Omron CX-Programmer project NewProject (CX-Programmer 9.75)

# PLC NewPLC1: CP1L M

## Global symbols (name address type ; comment)
0.00 BOOL  ; 灌装缸上限位
0.01 BOOL  ; 灌装缸下限位
0.02 BOOL  ; 缺瓶检测
0.03 BOOL  ; 出瓶检测
0.04 BOOL  ; 喷嘴检测
0.05 BOOL  ; 油嘴架上限位
0.06 BOOL  ; 油嘴架下限位
0.07 BOOL  ; 灌装缸原位
0.08 BOOL  ; 塞检测
0.09 BOOL  ; 中间堵瓶
0.10 BOOL  ; 星盘过载检测
0.11 BOOL  ; 星盘凸轮
100.02 BOOL  ; 进瓶阀门
100.03 BOOL  ; 出瓶阀门
100.04 BOOL  ; 夹瓶阀门
100.05 BOOL  ; 油嘴架阀门
100.06 BOOL  ; 吸盘上下阀门
100.07 BOOL  ; 吸盘前后阀门
101.00 BOOL  ; 输送带
101.01 BOOL  ; 星盘使能
101.02 BOOL  ; 真空阀门
101.03 BOOL  ; 敲塞阀门
101.04 BOOL  ; 剔除气缸
101.05 BOOL  ; 氮气阀门
1.00 BOOL  ; 门检测
1.01 BOOL  ; 加塞瓶检测
1.02 BOOL  ; 检测瓶检测
1.03 BOOL  ; 检测塞检测
1.04 BOOL  ; 剔除瓶检测
20.00 BOOL  ; 自动（触摸）
20.01 BOOL  ; 自动停（触摸）
20.04 BOOL  ; 单次灌装
20.05 BOOL  ; 灌装泵复位
20.06 BOOL  ; 装量修正
20.07 BOOL  ; 清除产量
21.00 BOOL  ; 进瓶手动
21.01 BOOL  ; 夹瓶手动
21.02 BOOL  ; 油嘴架手动
21.03 BOOL  ; 氮气手动
21.04 BOOL  ; 出瓶手动
21.05 BOOL  ; 输送带暂停
22.00 BOOL  ; 吸盘上下手动
22.01 BOOL  ; 真空手动
22.02 BOOL  ; 吸盘前后手动
22.03 BOOL  ; 敲塞手动
22.04 BOOL  ; 星盘点动
23.00 BOOL  ; 存参数
23.01 BOOL  ; 取参数
27.01 BOOL  ; 锁定
A280.04 BOOL  ; 灌装运行中
D100 CHANNEL  ; 上升加减速
D1000 CHANNEL  ; 产量
D1002 CHANNEL  ; 参数显示
D101 CHANNEL  ; 灌装上升速度
D110 CHANNEL  ; 下降加减速
D111 CHANNEL  ; 灌装缸下降速度
D120 CHANNEL  ; 复位加减速
D121 CHANNEL  ; 复位速度
D200 CHANNEL  ; 灌装脉冲数
D50 CHANNEL  ; 灌装次数
D600 CHANNEL  ; 1ml脉冲数
D6000 CHANNEL  ; 每圈装量
D6002 CHANNEL  ; 装量设定
D6003 CHANNEL  ; 实际装量
D6004 CHANNEL  ; 灌装缸上升速度
D6005 CHANNEL  ; 灌装缸下降速度
D6006 CHANNEL  ; 油嘴架延时上升
D6007 CHANNEL  ; 出瓶气缸关闭延时
D6008 CHANNEL  ; 进瓶气缸打开延时
D6009 CHANNEL  ; 灌装设定次数
D6010 CHANNEL  ; 吸盘上下延时设定
D6011 CHANNEL  ; 吸盘前/后延时设定
D6012 CHANNEL  ; 灌装头数设定
D604 CHANNEL  ; 总脉冲10倍
D608 CHANNEL  ; 总脉冲数
D612 CHANNEL  ; 实际每0.1ml脉冲数
D614 CHANNEL  ; 总脉冲10倍
D616 CHANNEL  ; 实际每圈装量
D650 CHANNEL  ; 灌装缸上升速度
D654 CHANNEL  ; 灌装缸上升速度
D660 CHANNEL  ; 灌装缸下降速度
D664 CHANNEL  ; 灌装缸下降速度
T0010 BOOL  ; 锁定时间
T0100 BOOL  ; 油嘴架下降延时
T0101 BOOL  ; 延时灌装
T0102 BOOL  ; 油嘴架延时上升
T0103 BOOL  ; 灌装结束延时
T0104 BOOL  ; 出瓶气缸延时打开
T0105 BOOL  ; 出瓶气缸关闭延时
T0106 BOOL  ; 进瓶气缸打开延时
T0107 BOOL  ; 灌装返回到位延时
T0108 BOOL  ; 进瓶气缸关闭延时
T0300 BOOL  ; 吸盘下延时
T0301 BOOL  ; 真空延时
T0302 BOOL  ; 吸盘上延时
T0303 BOOL  ; 吸盘前延时
T0304 BOOL  ; 吸盘下延时
T0305 BOOL  ; 真空释放延时
T0306 BOOL  ; 吸盘上延时
T0307 BOOL  ; 吸盘返回延时
T0500 BOOL  ; 剔除延时
W100.00 BOOL  ; 自动运行中
W100.01 BOOL  ; 停自动
W101.00 BOOL  ; 单次灌装中
W102.00 BOOL  ; 灌装泵复位中
W10.00 BOOL  ; 进瓶气缸
W10.01 BOOL  ; 夹瓶气缸
W10.02 BOOL  ; 油嘴架气缸
W10.03 BOOL  ; 氮气阀门
W10.04 BOOL  ; 出瓶气缸
W10.05 BOOL  ; 灌装泵
W200.00 BOOL  ; 星盘过载
W201.00 BOOL  ; 灌装缸上限位
W201.01 BOOL  ; 灌装缸下限位
W201.02 BOOL  ; 灌装缸原位异常
W201.03 BOOL  ; 油嘴架上限位
W201.04 BOOL  ; 油嘴架上限位
W201.05 BOOL  ; 油嘴架下限位
W201.06 BOOL  ; 灌装缸原位异常
W202.00 BOOL  ; 缺瓶报警
W202.01 BOOL  ; 中间堵瓶
W202.02 BOOL  ; 喷嘴异常
W203.00 BOOL  ; 出瓶堵
W203.01 BOOL  ; 门报警
W203.02 BOOL  ; 缺塞报警
W204.00 BOOL  ; 手动中
W204.01 BOOL  ; 自动中
W204.02 BOOL  ; 单次灌装中
W204.03 BOOL  ; 灌装泵复位中
W20.00 BOOL  ; 吸盘上下
W20.01 BOOL  ; 真空
W20.02 BOOL  ; 吸盘前后
W20.03 BOOL  ; 敲塞
W210.00 BOOL  ; 星盘过载
W210.01 BOOL  ; 灌装缸上限位
W210.02 BOOL  ; 灌装缸下限位
W210.03 BOOL  ; 灌装缸原位异常
W210.04 BOOL  ; 油嘴架上限位
W210.05 BOOL  ; 油嘴架下限位
W210.06 BOOL  ; 缺瓶报警
W210.07 BOOL  ; 中间堵瓶
W210.08 BOOL  ; 喷嘴异常
W211.00 BOOL  ; 出瓶堵
W211.01 BOOL  ; 门报警
W211.02 BOOL  ; 缺塞报警
W220.00 BOOL  ; 暂停报警条件
W220.01 BOOL  ; 灌装原位报警条件
W220.02 BOOL  ; 油嘴架上限位报警条件
W220.03 BOOL  ; 油嘴架上限位报警条件
W220.04 BOOL  ; 手动报警条件
W220.05 BOOL  ; 手动中
W220.06 BOOL  ; 自动报警条件
W220.07 BOOL  ; 单次灌装中报警条件
W220.08 BOOL  ; 灌装泵复位中报警条件
W3.00 BOOL  ; 停星盘中
W3.01 BOOL  ; 停星盘
W3.02 BOOL  ; 停自动停星盘中
W3.03 BOOL  ; 停自动停星盘
W3.04 BOOL  ; 点动停
W8.00 BOOL  ; 停输送带
出瓶堵 常开报警
单次灌装中 常开报警
灌装泵复位中 常开报警
灌装返回原位 常开报警
灌装缸上限 常闭报警
灌装缸下限 常闭报警
灌装缸原位 常闭报警
门报警 常闭报警
喷嘴异常 常闭报警
缺瓶报警 常闭报警
缺塞报警 常闭报警
手动中 常开报警
星盘过载 常开报警
油嘴架上限位 常闭报警
油嘴架上限位初始 常闭报警
油嘴架下限位 常开报警
中间堵瓶 常开报警
自动中 常开报警

## Program 新程序1 (cyclic task 0)

### Section 计算部分

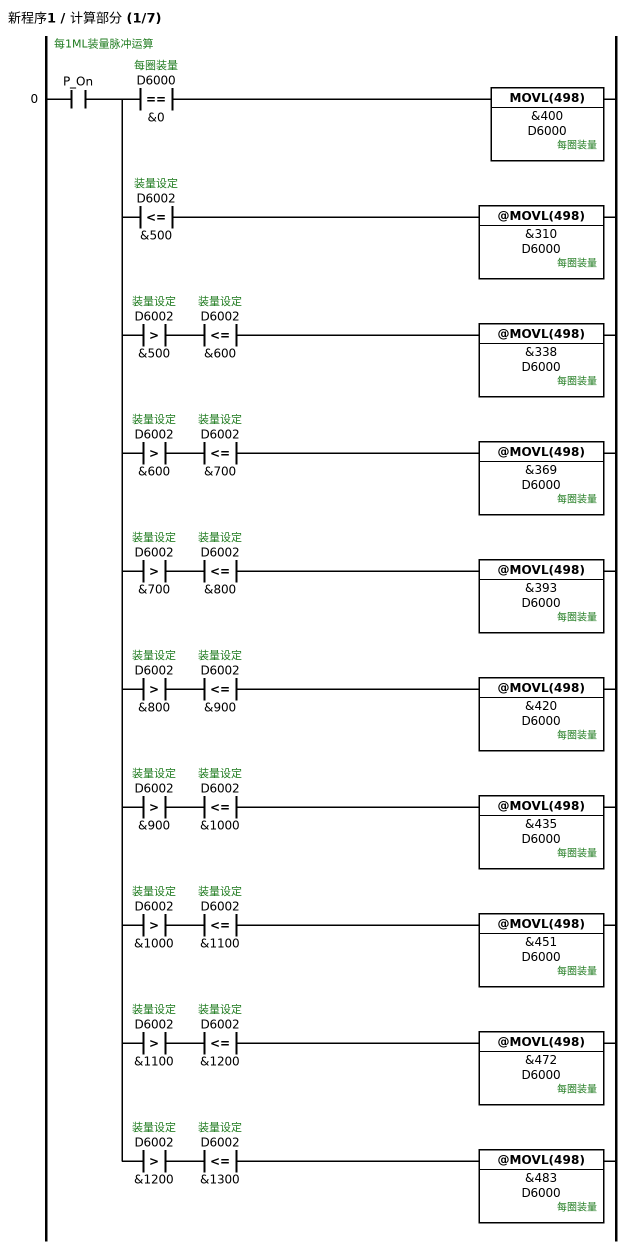
; rung 0: 每1ML装量脉冲运算
LD P_On
OUT TR0
AND=(300) D6000 &0  ; 每圈装量
MOVL(498) &400 D6000  ; 每圈装量
LD TR0
AND<=(315) D6002 &500  ; 装量设定
@MOVL(498) &310 D6000  ; 每圈装量
LD TR0
AND>(320) D6002 &500  ; 装量设定
AND<=(315) D6002 &600  ; 装量设定
@MOVL(498) &338 D6000  ; 每圈装量
LD TR0
AND>(320) D6002 &600  ; 装量设定
AND<=(315) D6002 &700  ; 装量设定
@MOVL(498) &369 D6000  ; 每圈装量
LD TR0
AND>(320) D6002 &700  ; 装量设定
AND<=(315) D6002 &800  ; 装量设定
@MOVL(498) &393 D6000  ; 每圈装量
LD TR0
AND>(320) D6002 &800  ; 装量设定
AND<=(315) D6002 &900  ; 装量设定
@MOVL(498) &420 D6000  ; 每圈装量
LD TR0
AND>(320) D6002 &900  ; 装量设定
AND<=(315) D6002 &1000  ; 装量设定
@MOVL(498) &435 D6000  ; 每圈装量
LD TR0
AND>(320) D6002 &1000  ; 装量设定
AND<=(315) D6002 &1100  ; 装量设定
@MOVL(498) &451 D6000  ; 每圈装量
LD TR0
AND>(320) D6002 &1100  ; 装量设定
AND<=(315) D6002 &1200  ; 装量设定
@MOVL(498) &472 D6000  ; 每圈装量
LD TR0
AND>(320) D6002 &1200  ; 装量设定
AND<=(315) D6002 &1300  ; 装量设定
@MOVL(498) &483 D6000  ; 每圈装量

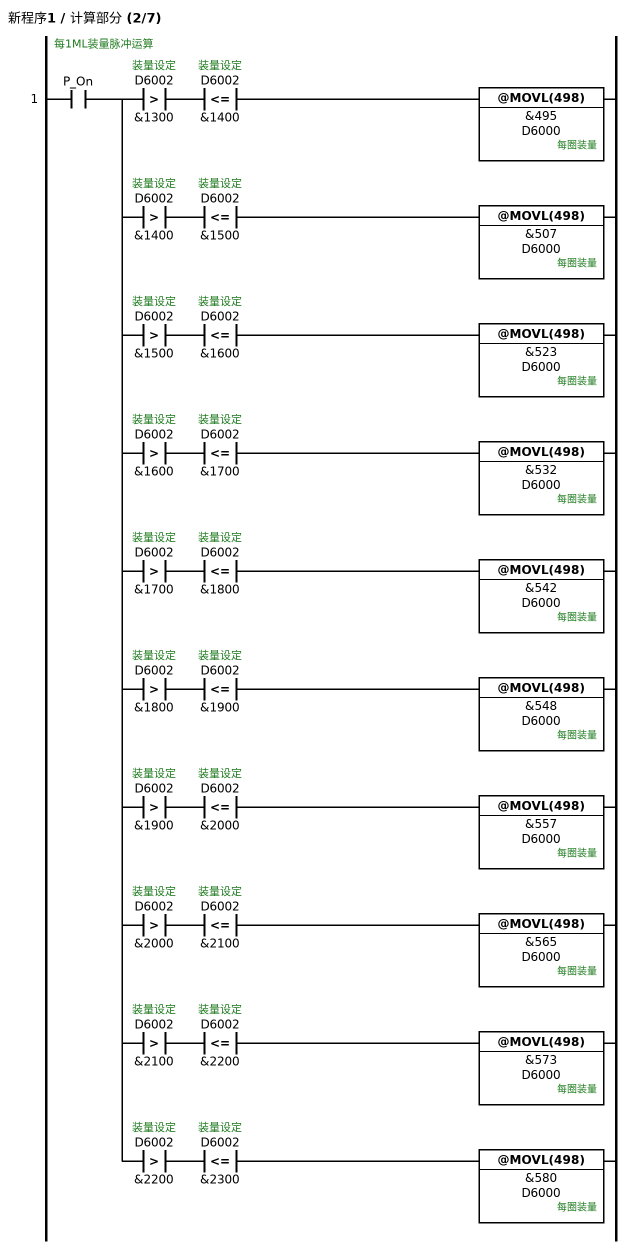
; rung 1: 每1ML装量脉冲运算
LD P_On
OUT TR0
AND>(320) D6002 &1300  ; 装量设定
AND<=(315) D6002 &1400  ; 装量设定
@MOVL(498) &495 D6000  ; 每圈装量
LD TR0
AND>(320) D6002 &1400  ; 装量设定
AND<=(315) D6002 &1500  ; 装量设定
@MOVL(498) &507 D6000  ; 每圈装量
LD TR0
AND>(320) D6002 &1500  ; 装量设定
AND<=(315) D6002 &1600  ; 装量设定
@MOVL(498) &523 D6000  ; 每圈装量
LD TR0
AND>(320) D6002 &1600  ; 装量设定
AND<=(315) D6002 &1700  ; 装量设定
@MOVL(498) &532 D6000  ; 每圈装量
LD TR0
AND>(320) D6002 &1700  ; 装量设定
AND<=(315) D6002 &1800  ; 装量设定
@MOVL(498) &542 D6000  ; 每圈装量
LD TR0
AND>(320) D6002 &1800  ; 装量设定
AND<=(315) D6002 &1900  ; 装量设定
@MOVL(498) &548 D6000  ; 每圈装量
LD TR0
AND>(320) D6002 &1900  ; 装量设定
AND<=(315) D6002 &2000  ; 装量设定
@MOVL(498) &557 D6000  ; 每圈装量
LD TR0
AND>(320) D6002 &2000  ; 装量设定
AND<=(315) D6002 &2100  ; 装量设定
@MOVL(498) &565 D6000  ; 每圈装量
LD TR0
AND>(320) D6002 &2100  ; 装量设定
AND<=(315) D6002 &2200  ; 装量设定
@MOVL(498) &573 D6000  ; 每圈装量
LD TR0
AND>(320) D6002 &2200  ; 装量设定
AND<=(315) D6002 &2300  ; 装量设定
@MOVL(498) &580 D6000  ; 每圈装量

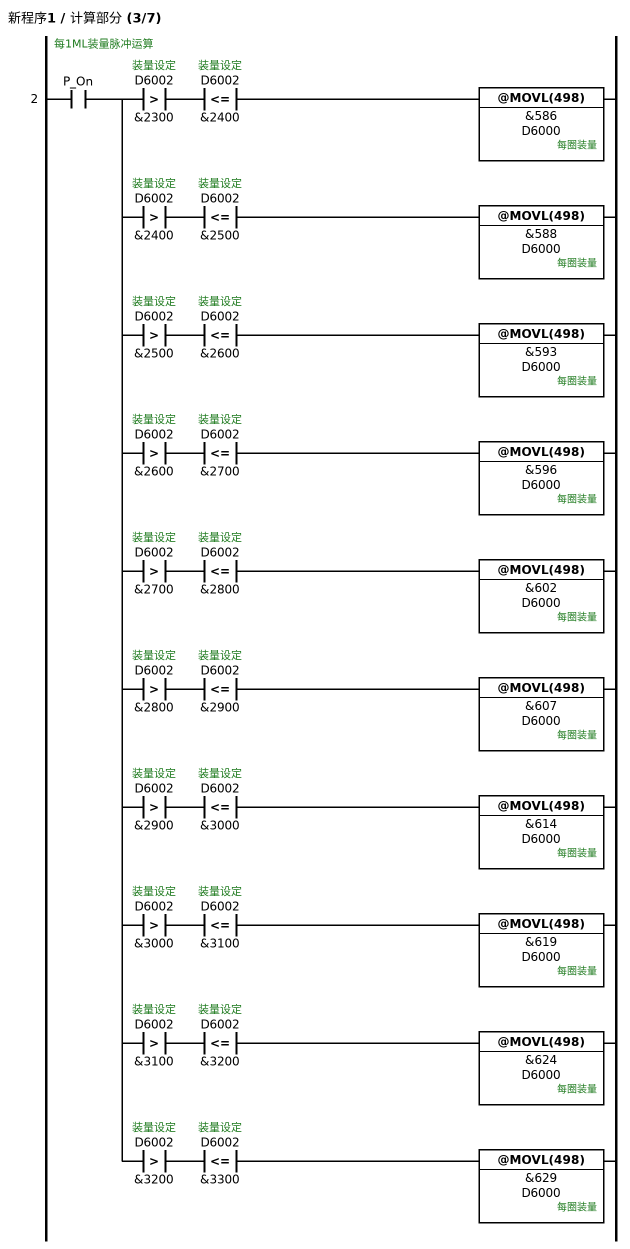
; rung 2: 每1ML装量脉冲运算
LD P_On
OUT TR0
AND>(320) D6002 &2300  ; 装量设定
AND<=(315) D6002 &2400  ; 装量设定
@MOVL(498) &586 D6000  ; 每圈装量
LD TR0
AND>(320) D6002 &2400  ; 装量设定
AND<=(315) D6002 &2500  ; 装量设定
@MOVL(498) &588 D6000  ; 每圈装量
LD TR0
AND>(320) D6002 &2500  ; 装量设定
AND<=(315) D6002 &2600  ; 装量设定
@MOVL(498) &593 D6000  ; 每圈装量
LD TR0
AND>(320) D6002 &2600  ; 装量设定
AND<=(315) D6002 &2700  ; 装量设定
@MOVL(498) &596 D6000  ; 每圈装量
LD TR0
AND>(320) D6002 &2700  ; 装量设定
AND<=(315) D6002 &2800  ; 装量设定
@MOVL(498) &602 D6000  ; 每圈装量
LD TR0
AND>(320) D6002 &2800  ; 装量设定
AND<=(315) D6002 &2900  ; 装量设定
@MOVL(498) &607 D6000  ; 每圈装量
LD TR0
AND>(320) D6002 &2900  ; 装量设定
AND<=(315) D6002 &3000  ; 装量设定
@MOVL(498) &614 D6000  ; 每圈装量
LD TR0
AND>(320) D6002 &3000  ; 装量设定
AND<=(315) D6002 &3100  ; 装量设定
@MOVL(498) &619 D6000  ; 每圈装量
LD TR0
AND>(320) D6002 &3100  ; 装量设定
AND<=(315) D6002 &3200  ; 装量设定
@MOVL(498) &624 D6000  ; 每圈装量
LD TR0
AND>(320) D6002 &3200  ; 装量设定
AND<=(315) D6002 &3300  ; 装量设定
@MOVL(498) &629 D6000  ; 每圈装量

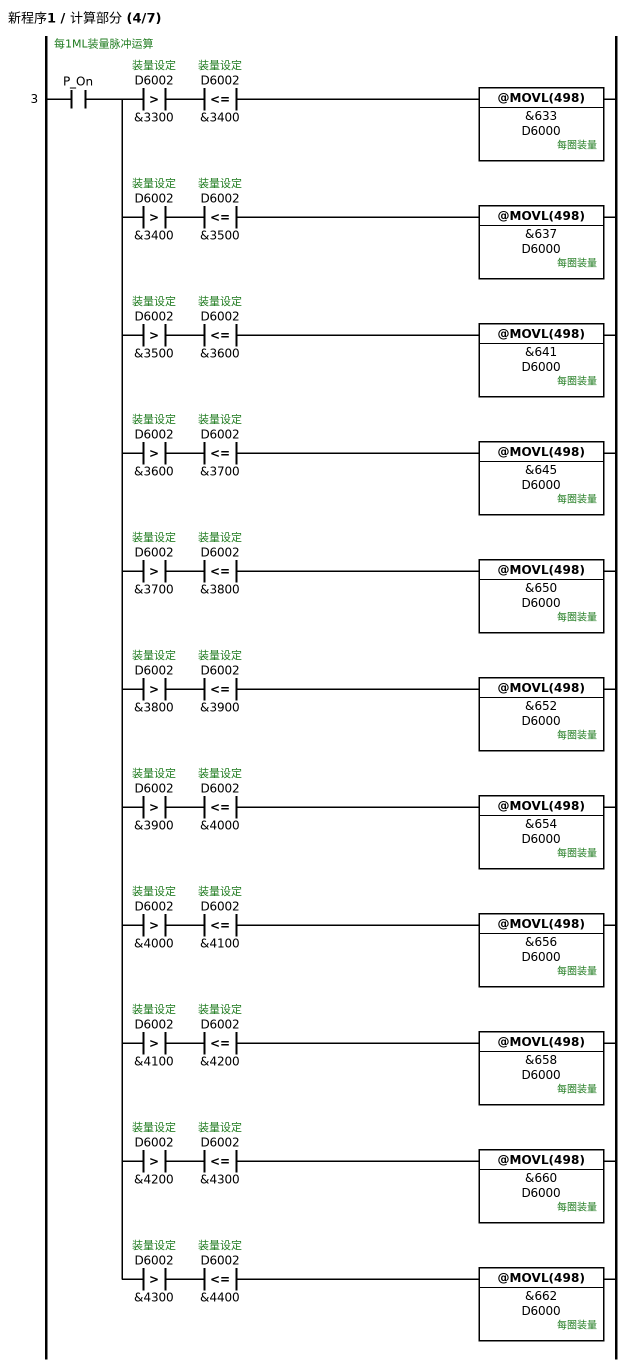
; rung 3: 每1ML装量脉冲运算
LD P_On
OUT TR0
AND>(320) D6002 &3300  ; 装量设定
AND<=(315) D6002 &3400  ; 装量设定
@MOVL(498) &633 D6000  ; 每圈装量
LD TR0
AND>(320) D6002 &3400  ; 装量设定
AND<=(315) D6002 &3500  ; 装量设定
@MOVL(498) &637 D6000  ; 每圈装量
LD TR0
AND>(320) D6002 &3500  ; 装量设定
AND<=(315) D6002 &3600  ; 装量设定
@MOVL(498) &641 D6000  ; 每圈装量
LD TR0
AND>(320) D6002 &3600  ; 装量设定
AND<=(315) D6002 &3700  ; 装量设定
@MOVL(498) &645 D6000  ; 每圈装量
LD TR0
AND>(320) D6002 &3700  ; 装量设定
AND<=(315) D6002 &3800  ; 装量设定
@MOVL(498) &650 D6000  ; 每圈装量
LD TR0
AND>(320) D6002 &3800  ; 装量设定
AND<=(315) D6002 &3900  ; 装量设定
@MOVL(498) &652 D6000  ; 每圈装量
LD TR0
AND>(320) D6002 &3900  ; 装量设定
AND<=(315) D6002 &4000  ; 装量设定
@MOVL(498) &654 D6000  ; 每圈装量
LD TR0
AND>(320) D6002 &4000  ; 装量设定
AND<=(315) D6002 &4100  ; 装量设定
@MOVL(498) &656 D6000  ; 每圈装量
LD TR0
AND>(320) D6002 &4100  ; 装量设定
AND<=(315) D6002 &4200  ; 装量设定
@MOVL(498) &658 D6000  ; 每圈装量
LD TR0
AND>(320) D6002 &4200  ; 装量设定
AND<=(315) D6002 &4300  ; 装量设定
@MOVL(498) &660 D6000  ; 每圈装量
LD TR0
AND>(320) D6002 &4300  ; 装量设定
AND<=(315) D6002 &4400  ; 装量设定
@MOVL(498) &662 D6000  ; 每圈装量

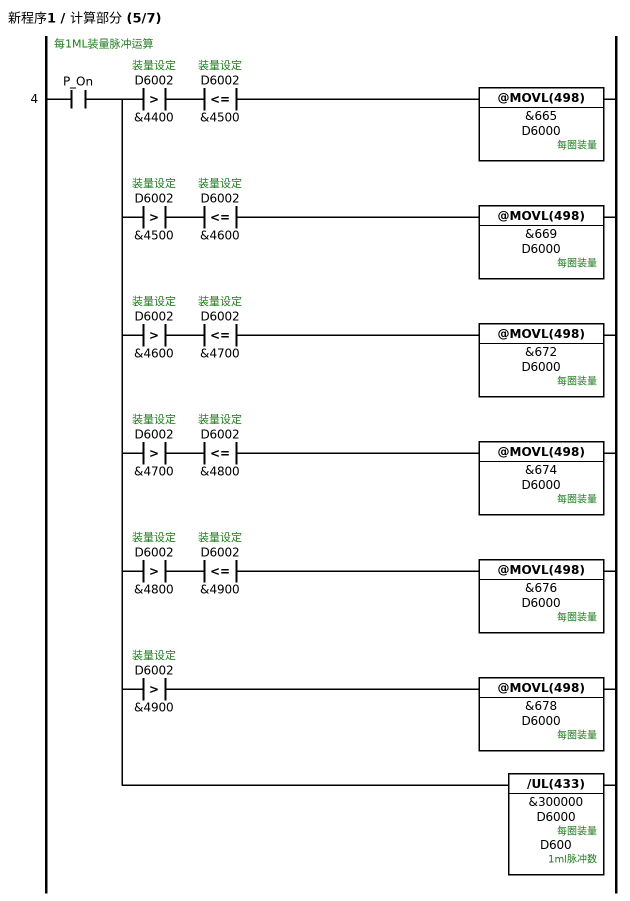
; rung 4: 每1ML装量脉冲运算
LD P_On
OUT TR0
AND>(320) D6002 &4400  ; 装量设定
AND<=(315) D6002 &4500  ; 装量设定
@MOVL(498) &665 D6000  ; 每圈装量
LD TR0
AND>(320) D6002 &4500  ; 装量设定
AND<=(315) D6002 &4600  ; 装量设定
@MOVL(498) &669 D6000  ; 每圈装量
LD TR0
AND>(320) D6002 &4600  ; 装量设定
AND<=(315) D6002 &4700  ; 装量设定
@MOVL(498) &672 D6000  ; 每圈装量
LD TR0
AND>(320) D6002 &4700  ; 装量设定
AND<=(315) D6002 &4800  ; 装量设定
@MOVL(498) &674 D6000  ; 每圈装量
LD TR0
AND>(320) D6002 &4800  ; 装量设定
AND<=(315) D6002 &4900  ; 装量设定
@MOVL(498) &676 D6000  ; 每圈装量
LD TR0
AND>(320) D6002 &4900  ; 装量设定
@MOVL(498) &678 D6000  ; 每圈装量
LD TR0
/UL(433) &300000 D6000 D600  ; 每圈装量, 1ml脉冲数

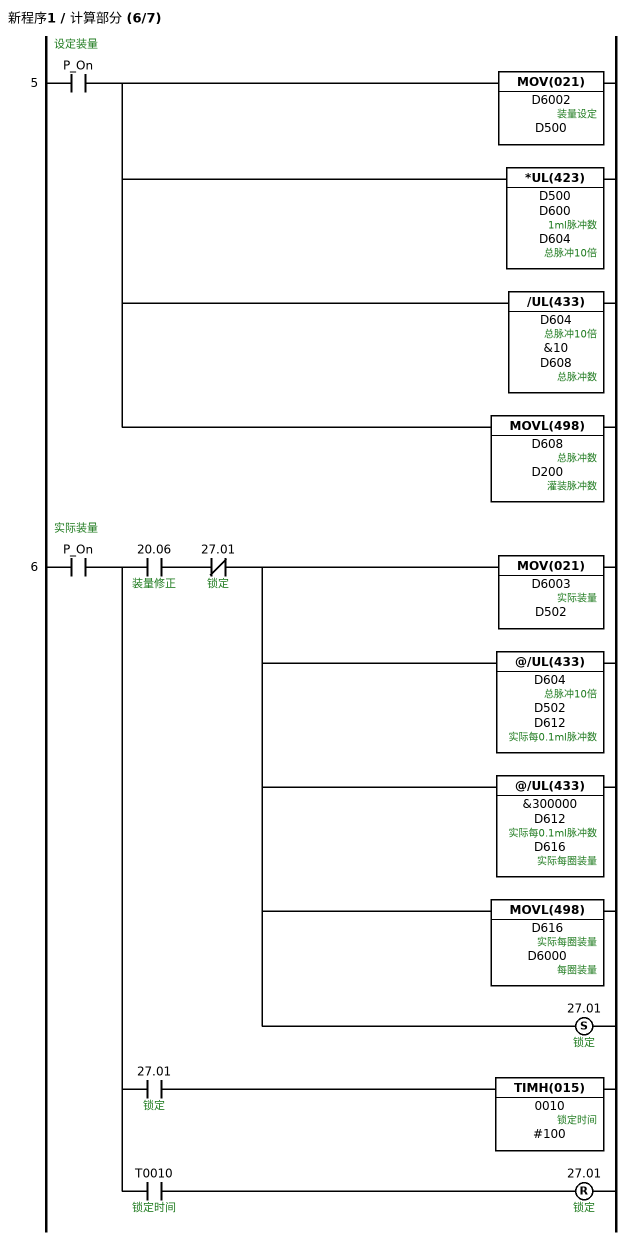
; rung 5: 设定装量
LD P_On
MOV(021) D6002 D500  ; 装量设定
*UL(423) D500 D600 D604  ; 1ml脉冲数, 总脉冲10倍
/UL(433) D604 &10 D608  ; 总脉冲10倍, 总脉冲数
MOVL(498) D608 D200  ; 总脉冲数, 灌装脉冲数
; rung 6: 实际装量
LD P_On
OUT TR0
AND 20.06  ; 装量修正
ANDNOT 27.01  ; 锁定
MOV(021) D6003 D502  ; 实际装量
@/UL(433) D604 D502 D612  ; 总脉冲10倍, 实际每0.1ml脉冲数
@/UL(433) &300000 D612 D616  ; 实际每0.1ml脉冲数, 实际每圈装量
MOVL(498) D616 D6000  ; 实际每圈装量, 每圈装量
SET 27.01  ; 锁定
LD TR0
AND 27.01  ; 锁定
TIMH(015) 0010 #100  ; 锁定时间
LD TR0
AND T0010  ; 锁定时间
RSET 27.01  ; 锁定

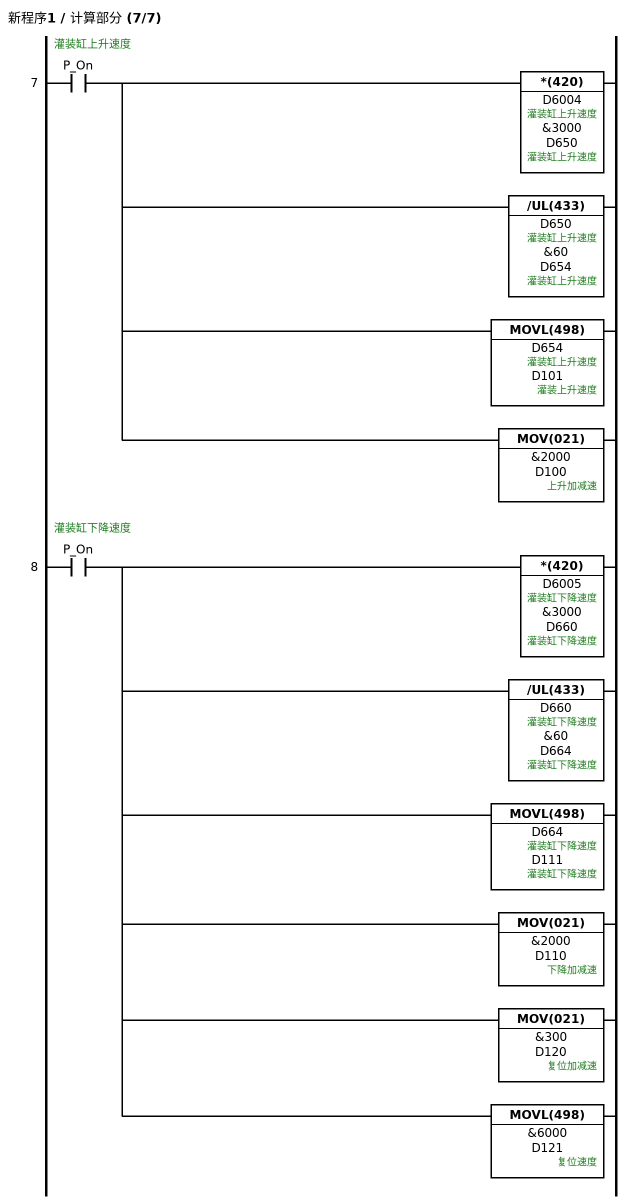
; rung 7: 灌装缸上升速度
LD P_On
*(420) D6004 &3000 D650  ; 灌装缸上升速度
/UL(433) D650 &60 D654  ; 灌装缸上升速度
MOVL(498) D654 D101  ; 灌装缸上升速度, 灌装上升速度
MOV(021) &2000 D100  ; 上升加减速
; rung 8: 灌装缸下降速度
LD P_On
*(420) D6005 &3000 D660  ; 灌装缸下降速度
/UL(433) D660 &60 D664  ; 灌装缸下降速度
MOVL(498) D664 D111  ; 灌装缸下降速度
MOV(021) &2000 D110  ; 下降加减速
MOV(021) &300 D120  ; 复位加减速
MOVL(498) &6000 D121  ; 复位速度

### Section 控制部分

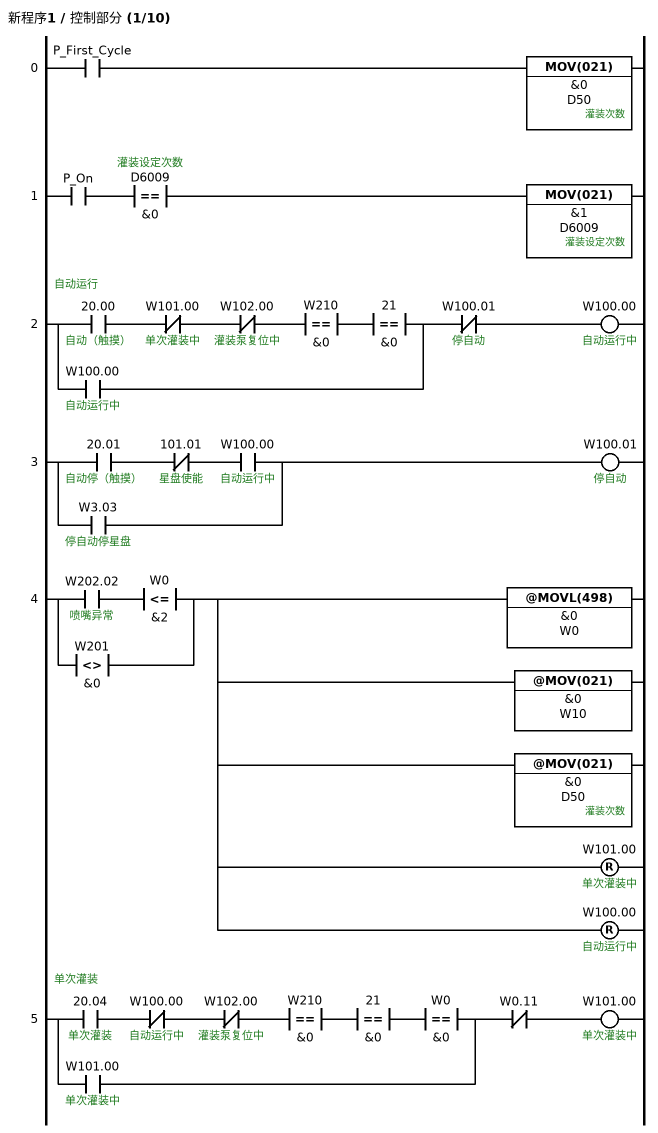
; rung 0
LD P_First_Cycle
MOV(021) &0 D50  ; 灌装次数
; rung 1
LD P_On
AND=(300) D6009 &0  ; 灌装设定次数
MOV(021) &1 D6009  ; 灌装设定次数
; rung 2: 自动运行
LD 20.00  ; 自动（触摸）
ANDNOT W101.00  ; 单次灌装中
ANDNOT W102.00  ; 灌装泵复位中
AND=L(301) W210 &0
AND=L(301) 21 &0
OR W100.00  ; 自动运行中
ANDNOT W100.01  ; 停自动
OUT W100.00  ; 自动运行中
; rung 3
LD 20.01  ; 自动停（触摸）
ANDNOT 101.01  ; 星盘使能
AND W100.00  ; 自动运行中
OR W3.03  ; 停自动停星盘
OUT W100.01  ; 停自动
; rung 4
LD W202.02  ; 喷嘴异常
AND<=(315) W0 &2
OR<>(305) W201 &0
@MOVL(498) &0 W0
@MOV(021) &0 W10
@MOV(021) &0 D50  ; 灌装次数
RSET W101.00  ; 单次灌装中
RSET W100.00  ; 自动运行中
; rung 5: 单次灌装
LD 20.04  ; 单次灌装
ANDNOT W100.00  ; 自动运行中
ANDNOT W102.00  ; 灌装泵复位中
AND=(300) W210 &0
AND=(300) 21 &0
AND=L(301) W0 &0
OR W101.00  ; 单次灌装中
ANDNOT W0.11
OUT W101.00  ; 单次灌装中

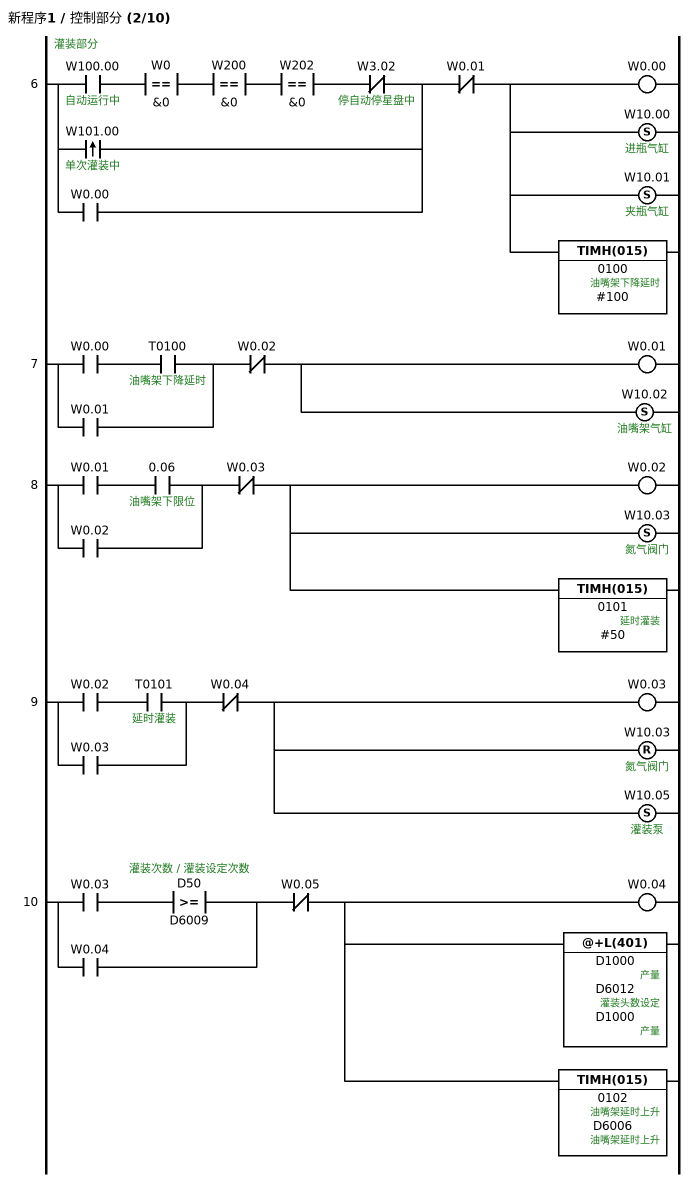
; rung 6: 灌装部分
LD W100.00  ; 自动运行中
AND=(300) W0 &0
AND=L(301) W200 &0
AND=(300) W202 &0
ANDNOT W3.02  ; 停自动停星盘中
@OR W101.00  ; 单次灌装中
OR W0.00
ANDNOT W0.01
OUT W0.00
SET W10.00  ; 进瓶气缸
SET W10.01  ; 夹瓶气缸
TIMH(015) 0100 #100  ; 油嘴架下降延时
; rung 7
LD W0.00
AND T0100  ; 油嘴架下降延时
OR W0.01
ANDNOT W0.02
OUT W0.01
SET W10.02  ; 油嘴架气缸
; rung 8
LD W0.01
AND 0.06  ; 油嘴架下限位
OR W0.02
ANDNOT W0.03
OUT W0.02
SET W10.03  ; 氮气阀门
TIMH(015) 0101 #50  ; 延时灌装
; rung 9
LD W0.02
AND T0101  ; 延时灌装
OR W0.03
ANDNOT W0.04
OUT W0.03
RSET W10.03  ; 氮气阀门
SET W10.05  ; 灌装泵
; rung 10
LD W0.03
AND>=(325) D50 D6009  ; 灌装次数, 灌装设定次数
OR W0.04
ANDNOT W0.05
OUT W0.04
@+L(401) D1000 D6012 D1000  ; 产量, 灌装头数设定
TIMH(015) 0102 D6006  ; 油嘴架延时上升

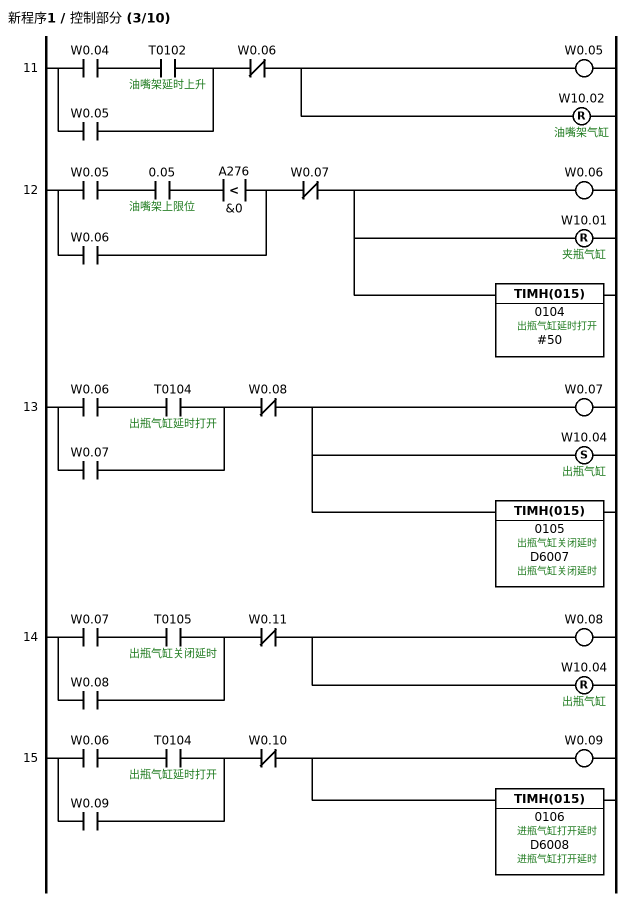
; rung 11
LD W0.04
AND T0102  ; 油嘴架延时上升
OR W0.05
ANDNOT W0.06
OUT W0.05
RSET W10.02  ; 油嘴架气缸
; rung 12
LD W0.05
AND 0.05  ; 油嘴架上限位
AND<SL(313) A276 &0
OR W0.06
ANDNOT W0.07
OUT W0.06
RSET W10.01  ; 夹瓶气缸
TIMH(015) 0104 #50  ; 出瓶气缸延时打开
; rung 13
LD W0.06
AND T0104  ; 出瓶气缸延时打开
OR W0.07
ANDNOT W0.08
OUT W0.07
SET W10.04  ; 出瓶气缸
TIMH(015) 0105 D6007  ; 出瓶气缸关闭延时
; rung 14
LD W0.07
AND T0105  ; 出瓶气缸关闭延时
OR W0.08
ANDNOT W0.11
OUT W0.08
RSET W10.04  ; 出瓶气缸
; rung 15
LD W0.06
AND T0104  ; 出瓶气缸延时打开
OR W0.09
ANDNOT W0.10
OUT W0.09
TIMH(015) 0106 D6008  ; 进瓶气缸打开延时

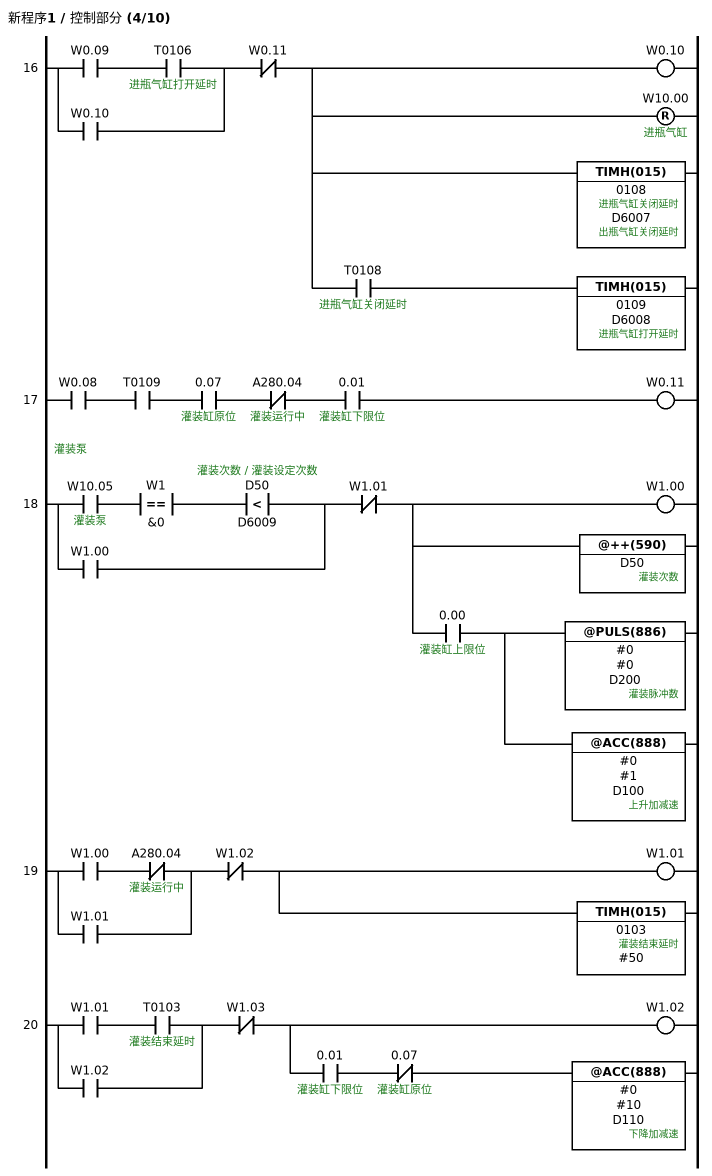
; rung 16
LD W0.09
AND T0106  ; 进瓶气缸打开延时
OR W0.10
ANDNOT W0.11
OUT W0.10
RSET W10.00  ; 进瓶气缸
TIMH(015) 0108 D6007  ; 出瓶气缸关闭延时, 进瓶气缸关闭延时
AND T0108  ; 进瓶气缸关闭延时
TIMH(015) 0109 D6008  ; 进瓶气缸打开延时
; rung 17
LD W0.08
AND T0109
AND 0.07  ; 灌装缸原位
ANDNOT A280.04  ; 灌装运行中
AND 0.01  ; 灌装缸下限位
OUT W0.11
; rung 18: 灌装泵
LD W10.05  ; 灌装泵
AND=(300) W1 &0
AND<(310) D50 D6009  ; 灌装次数, 灌装设定次数
OR W1.00
ANDNOT W1.01
OUT W1.00
@++(590) D50  ; 灌装次数
AND 0.00  ; 灌装缸上限位
@PULS(886) #0 #0 D200  ; 灌装脉冲数
@ACC(888) #0 #1 D100  ; 上升加减速
; rung 19
LD W1.00
ANDNOT A280.04  ; 灌装运行中
OR W1.01
ANDNOT W1.02
OUT W1.01
TIMH(015) 0103 #50  ; 灌装结束延时
; rung 20
LD W1.01
AND T0103  ; 灌装结束延时
OR W1.02
ANDNOT W1.03
OUT W1.02
AND 0.01  ; 灌装缸下限位
ANDNOT 0.07  ; 灌装缸原位
@ACC(888) #0 #10 D110  ; 下降加减速

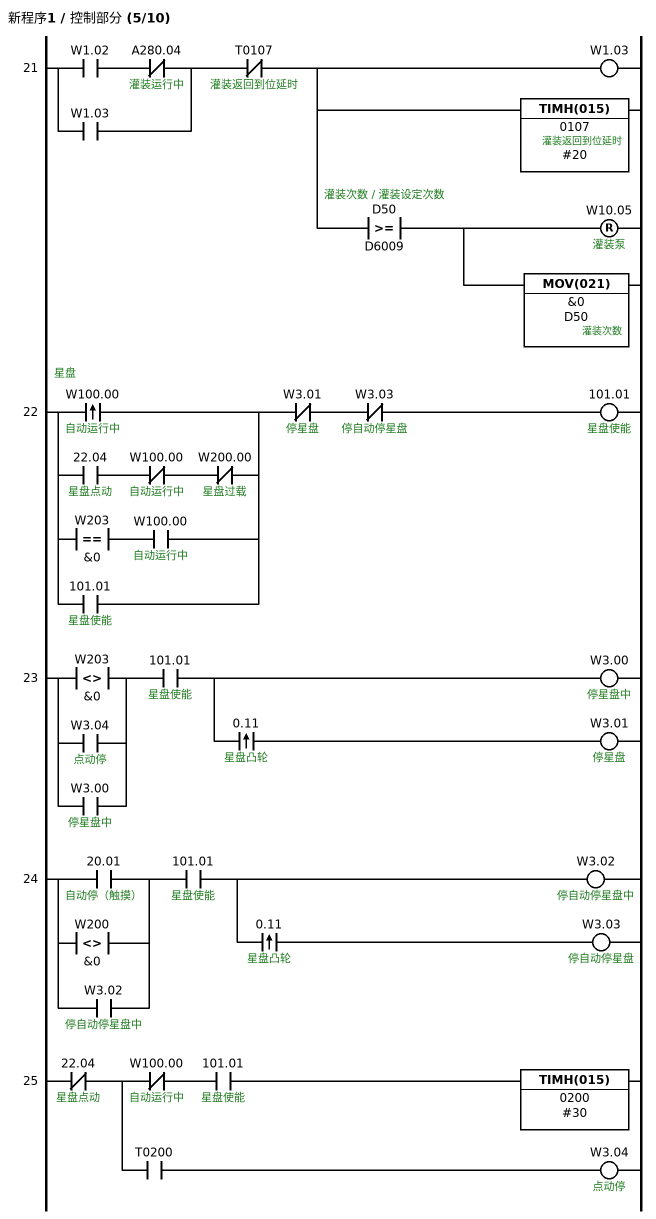
; rung 21
LD W1.02
ANDNOT A280.04  ; 灌装运行中
OR W1.03
ANDNOT T0107  ; 灌装返回到位延时
OUT W1.03
TIMH(015) 0107 #20  ; 灌装返回到位延时
AND>=(325) D50 D6009  ; 灌装次数, 灌装设定次数
RSET W10.05  ; 灌装泵
MOV(021) &0 D50  ; 灌装次数
; rung 22: 星盘
@LD W100.00  ; 自动运行中
LD 22.04  ; 星盘点动
ANDNOT W100.00  ; 自动运行中
ANDNOT W200.00  ; 星盘过载
ORLD
LD=(300) W203 &0
AND W100.00  ; 自动运行中
ORLD
OR 101.01  ; 星盘使能
ANDNOT W3.01  ; 停星盘
ANDNOT W3.03  ; 停自动停星盘
OUT 101.01  ; 星盘使能
; rung 23
LD<>(305) W203 &0
OR W3.04  ; 点动停
OR W3.00  ; 停星盘中
AND 101.01  ; 星盘使能
OUT W3.00  ; 停星盘中
@AND 0.11  ; 星盘凸轮
OUT W3.01  ; 停星盘
; rung 24
LD 20.01  ; 自动停（触摸）
OR<>L(306) W200 &0
OR W3.02  ; 停自动停星盘中
AND 101.01  ; 星盘使能
OUT W3.02  ; 停自动停星盘中
@AND 0.11  ; 星盘凸轮
OUT W3.03  ; 停自动停星盘
; rung 25
LDNOT 22.04  ; 星盘点动
OUT TR0
ANDNOT W100.00  ; 自动运行中
AND 101.01  ; 星盘使能
TIMH(015) 0200 #30
LD TR0
AND T0200
OUT W3.04  ; 点动停

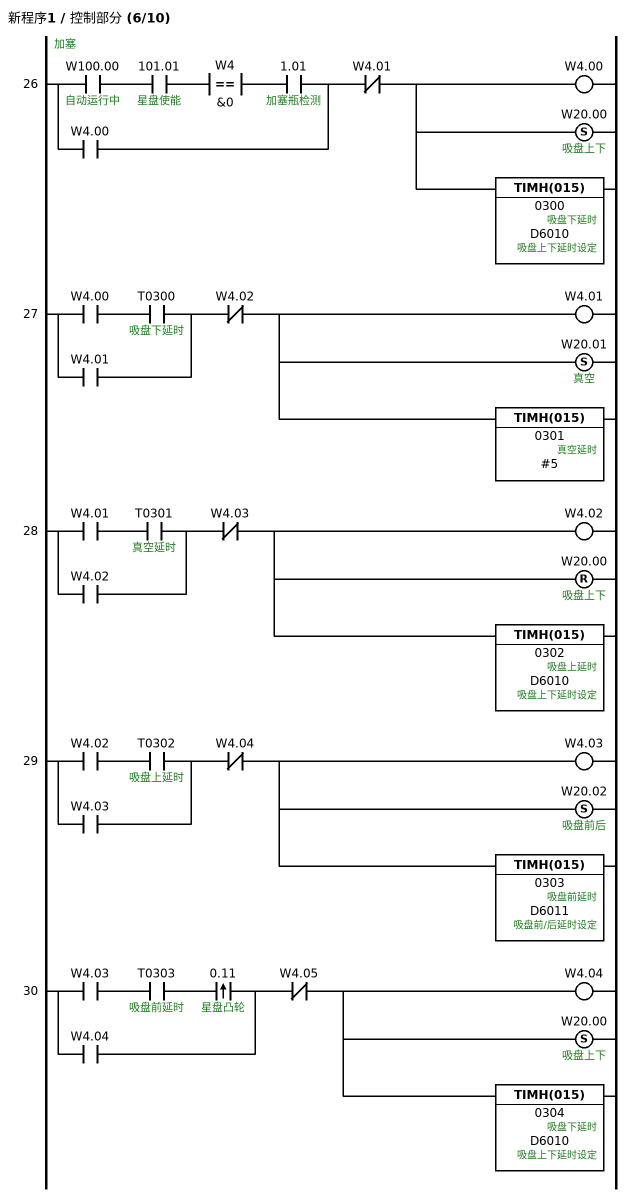
; rung 26: 加塞
LD W100.00  ; 自动运行中
AND 101.01  ; 星盘使能
AND=(300) W4 &0
AND 1.01  ; 加塞瓶检测
OR W4.00
ANDNOT W4.01
OUT W4.00
SET W20.00  ; 吸盘上下
TIMH(015) 0300 D6010  ; 吸盘上下延时设定, 吸盘下延时
; rung 27
LD W4.00
AND T0300  ; 吸盘下延时
OR W4.01
ANDNOT W4.02
OUT W4.01
SET W20.01  ; 真空
TIMH(015) 0301 #5  ; 真空延时
; rung 28
LD W4.01
AND T0301  ; 真空延时
OR W4.02
ANDNOT W4.03
OUT W4.02
RSET W20.00  ; 吸盘上下
TIMH(015) 0302 D6010  ; 吸盘上下延时设定, 吸盘上延时
; rung 29
LD W4.02
AND T0302  ; 吸盘上延时
OR W4.03
ANDNOT W4.04
OUT W4.03
SET W20.02  ; 吸盘前后
TIMH(015) 0303 D6011  ; 吸盘前/后延时设定, 吸盘前延时
; rung 30
LD W4.03
AND T0303  ; 吸盘前延时
@AND 0.11  ; 星盘凸轮
OR W4.04
ANDNOT W4.05
OUT W4.04
SET W20.00  ; 吸盘上下
TIMH(015) 0304 D6010  ; 吸盘上下延时设定, 吸盘下延时

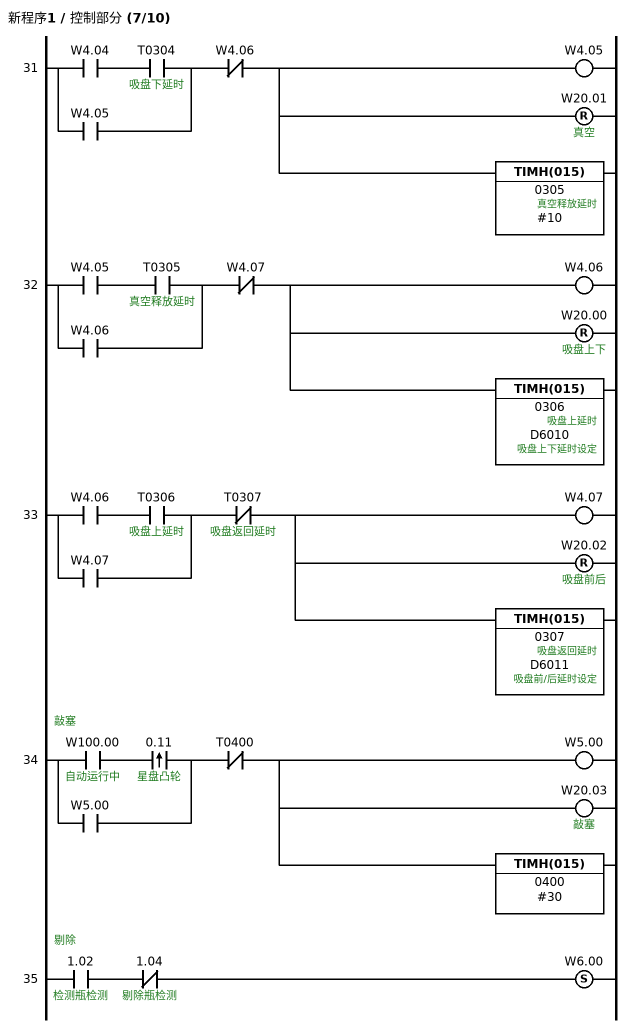
; rung 31
LD W4.04
AND T0304  ; 吸盘下延时
OR W4.05
ANDNOT W4.06
OUT W4.05
RSET W20.01  ; 真空
TIMH(015) 0305 #10  ; 真空释放延时
; rung 32
LD W4.05
AND T0305  ; 真空释放延时
OR W4.06
ANDNOT W4.07
OUT W4.06
RSET W20.00  ; 吸盘上下
TIMH(015) 0306 D6010  ; 吸盘上下延时设定, 吸盘上延时
; rung 33
LD W4.06
AND T0306  ; 吸盘上延时
OR W4.07
ANDNOT T0307  ; 吸盘返回延时
OUT W4.07
RSET W20.02  ; 吸盘前后
TIMH(015) 0307 D6011  ; 吸盘前/后延时设定, 吸盘返回延时
; rung 34: 敲塞
LD W100.00  ; 自动运行中
@AND 0.11  ; 星盘凸轮
OR W5.00
ANDNOT T0400
OUT W5.00
OUT W20.03  ; 敲塞
TIMH(015) 0400 #30
; rung 35: 剔除
LD 1.02  ; 检测瓶检测
ANDNOT 1.04  ; 剔除瓶检测
SET W6.00

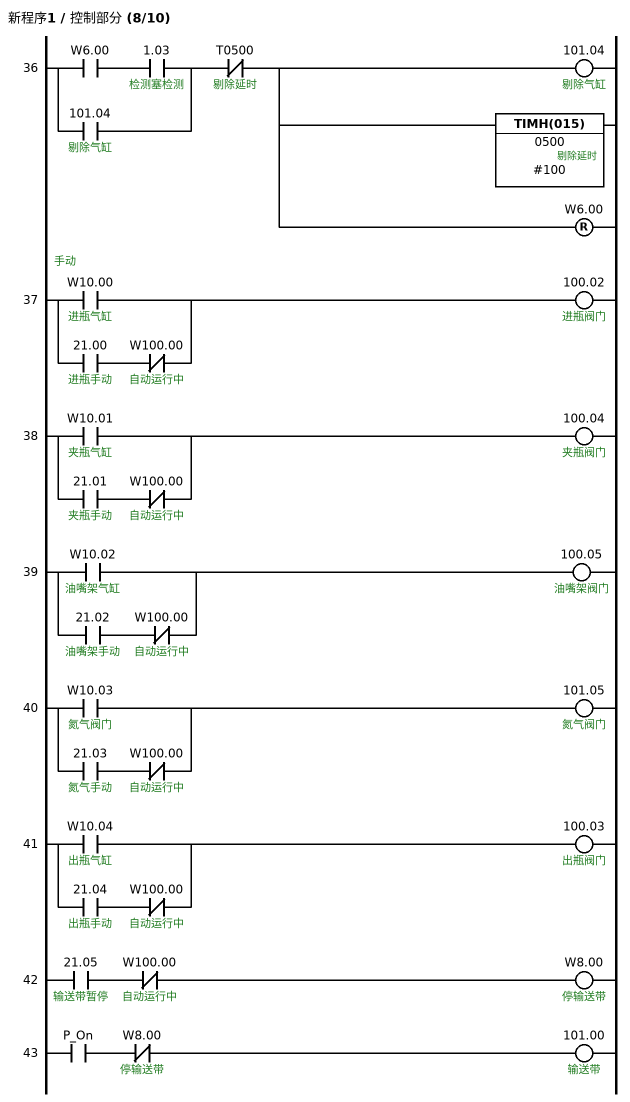
; rung 36
LD W6.00
AND 1.03  ; 检测塞检测
OR 101.04  ; 剔除气缸
ANDNOT T0500  ; 剔除延时
OUT 101.04  ; 剔除气缸
TIMH(015) 0500 #100  ; 剔除延时
RSET W6.00
; rung 37: 手动
LD W10.00  ; 进瓶气缸
LD 21.00  ; 进瓶手动
ANDNOT W100.00  ; 自动运行中
ORLD
OUT 100.02  ; 进瓶阀门
; rung 38
LD W10.01  ; 夹瓶气缸
LD 21.01  ; 夹瓶手动
ANDNOT W100.00  ; 自动运行中
ORLD
OUT 100.04  ; 夹瓶阀门
; rung 39
LD W10.02  ; 油嘴架气缸
LD 21.02  ; 油嘴架手动
ANDNOT W100.00  ; 自动运行中
ORLD
OUT 100.05  ; 油嘴架阀门
; rung 40
LD W10.03  ; 氮气阀门
LD 21.03  ; 氮气手动
ANDNOT W100.00  ; 自动运行中
ORLD
OUT 101.05  ; 氮气阀门
; rung 41
LD W10.04  ; 出瓶气缸
LD 21.04  ; 出瓶手动
ANDNOT W100.00  ; 自动运行中
ORLD
OUT 100.03  ; 出瓶阀门
; rung 42
LD 21.05  ; 输送带暂停
ANDNOT W100.00  ; 自动运行中
OUT W8.00  ; 停输送带
; rung 43
LD P_On
ANDNOT W8.00  ; 停输送带
OUT 101.00  ; 输送带

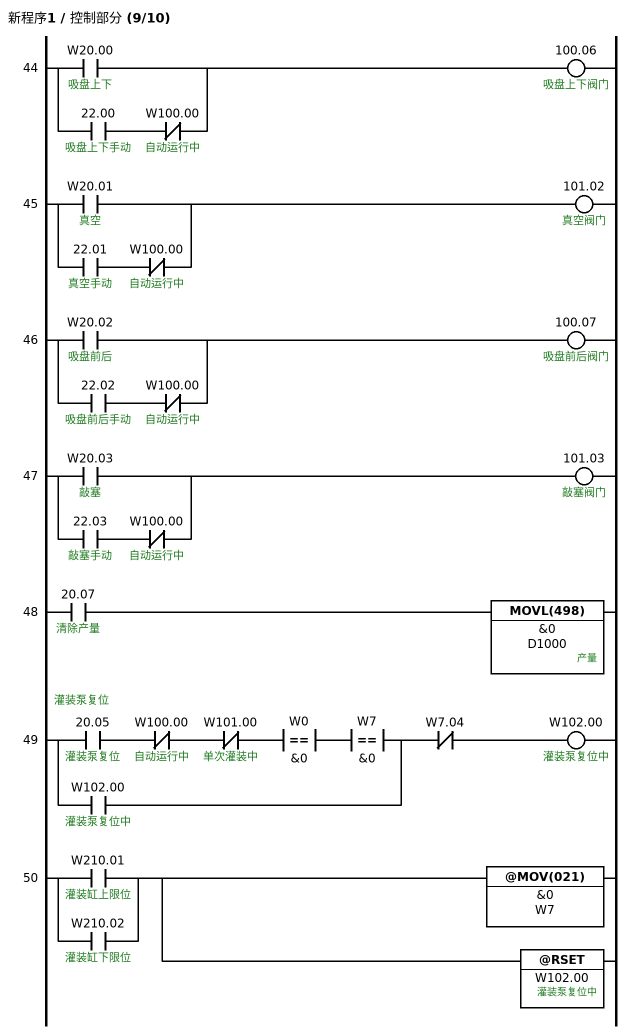
; rung 44
LD W20.00  ; 吸盘上下
LD 22.00  ; 吸盘上下手动
ANDNOT W100.00  ; 自动运行中
ORLD
OUT 100.06  ; 吸盘上下阀门
; rung 45
LD W20.01  ; 真空
LD 22.01  ; 真空手动
ANDNOT W100.00  ; 自动运行中
ORLD
OUT 101.02  ; 真空阀门
; rung 46
LD W20.02  ; 吸盘前后
LD 22.02  ; 吸盘前后手动
ANDNOT W100.00  ; 自动运行中
ORLD
OUT 100.07  ; 吸盘前后阀门
; rung 47
LD W20.03  ; 敲塞
LD 22.03  ; 敲塞手动
ANDNOT W100.00  ; 自动运行中
ORLD
OUT 101.03  ; 敲塞阀门
; rung 48
LD 20.07  ; 清除产量
MOVL(498) &0 D1000  ; 产量
; rung 49: 灌装泵复位
LD 20.05  ; 灌装泵复位
ANDNOT W100.00  ; 自动运行中
ANDNOT W101.00  ; 单次灌装中
AND=L(301) W0 &0
AND=(300) W7 &0
OR W102.00  ; 灌装泵复位中
ANDNOT W7.04
OUT W102.00  ; 灌装泵复位中
; rung 50
LD W210.01  ; 灌装缸上限位
OR W210.02  ; 灌装缸下限位
@MOV(021) &0 W7
@RSET W102.00  ; 灌装泵复位中

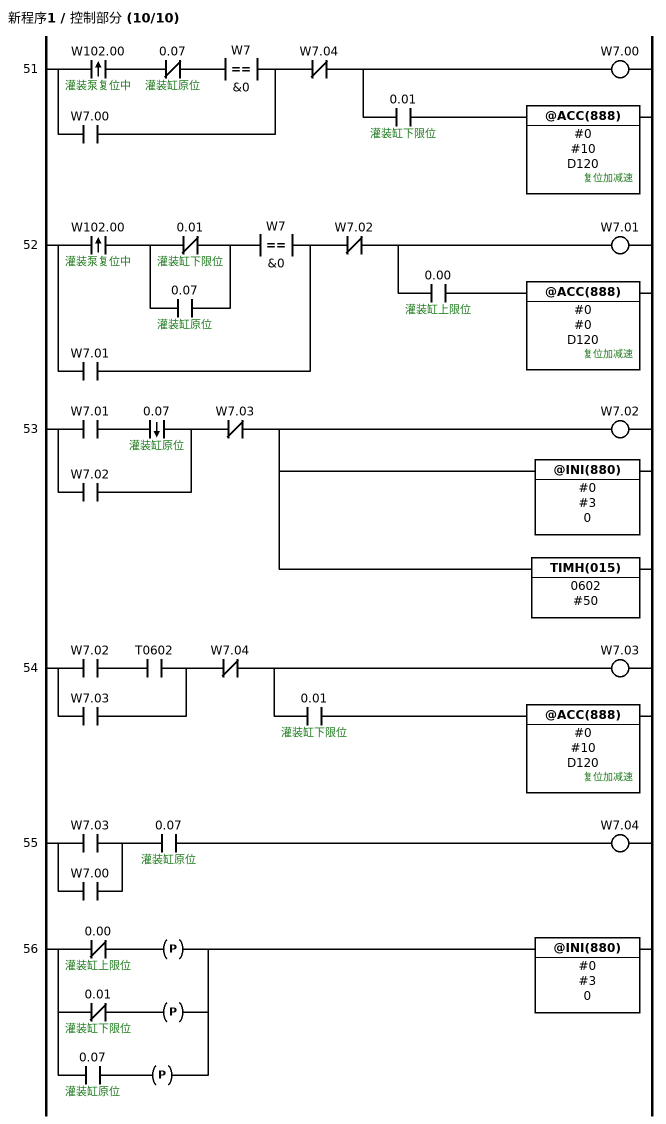
; rung 51
@LD W102.00  ; 灌装泵复位中
ANDNOT 0.07  ; 灌装缸原位
AND=(300) W7 &0
OR W7.00
ANDNOT W7.04
OUT W7.00
AND 0.01  ; 灌装缸下限位
@ACC(888) #0 #10 D120  ; 复位加减速
; rung 52
@LD W102.00  ; 灌装泵复位中
LDNOT 0.01  ; 灌装缸下限位
OR 0.07  ; 灌装缸原位
ANDLD
AND=(300) W7 &0
OR W7.01
ANDNOT W7.02
OUT W7.01
AND 0.00  ; 灌装缸上限位
@ACC(888) #0 #0 D120  ; 复位加减速
; rung 53
LD W7.01
%AND 0.07  ; 灌装缸原位
OR W7.02
ANDNOT W7.03
OUT W7.02
@INI(880) #0 #3 0
TIMH(015) 0602 #50
; rung 54
LD W7.02
AND T0602
OR W7.03
ANDNOT W7.04
OUT W7.03
AND 0.01  ; 灌装缸下限位
@ACC(888) #0 #10 D120  ; 复位加减速
; rung 55
LD W7.03
OR W7.00
AND 0.07  ; 灌装缸原位
OUT W7.04
; rung 56
LDNOT 0.00  ; 灌装缸上限位
UP(521)
LDNOT 0.01  ; 灌装缸下限位
UP(521)
ORLD
LD 0.07  ; 灌装缸原位
UP(521)
ORLD
@INI(880) #0 #3 0

### Section 报警部分

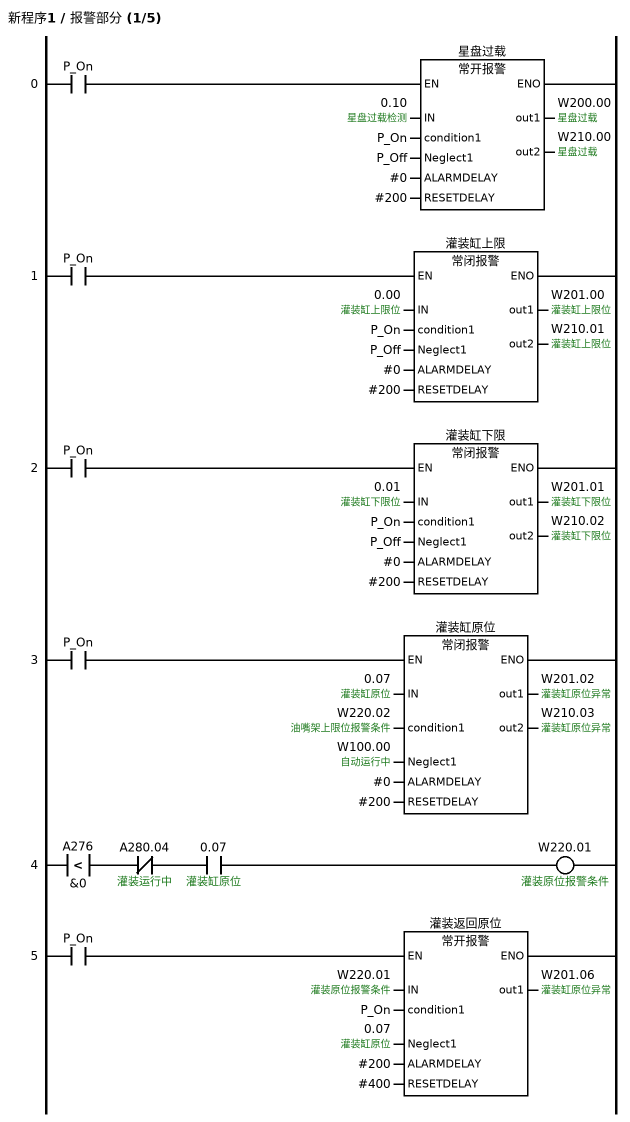
; rung 0
LD P_On
CALL 星盘过载 : 常开报警 (IN := 0.10, condition1 := P_On, Neglect1 := P_Off, ALARMDELAY := #0, RESETDELAY := #200, out1 => W200.00, out2 => W210.00)  ; 星盘过载检测, 星盘过载
; rung 1
LD P_On
CALL 灌装缸上限 : 常闭报警 (IN := 0.00, condition1 := P_On, Neglect1 := P_Off, ALARMDELAY := #0, RESETDELAY := #200, out1 => W201.00, out2 => W210.01)  ; 灌装缸上限位
; rung 2
LD P_On
CALL 灌装缸下限 : 常闭报警 (IN := 0.01, condition1 := P_On, Neglect1 := P_Off, ALARMDELAY := #0, RESETDELAY := #200, out1 => W201.01, out2 => W210.02)  ; 灌装缸下限位
; rung 3
LD P_On
CALL 灌装缸原位 : 常闭报警 (IN := 0.07, condition1 := W220.02, Neglect1 := W100.00, ALARMDELAY := #0, RESETDELAY := #200, out1 => W201.02, out2 => W210.03)  ; 灌装缸原位, 油嘴架上限位报警条件, 自动运行中, 灌装缸原位异常
; rung 4
LD<SL(313) A276 &0
ANDNOT A280.04  ; 灌装运行中
AND 0.07  ; 灌装缸原位
OUT W220.01  ; 灌装原位报警条件
; rung 5
LD P_On
CALL 灌装返回原位 : 常开报警 (IN := W220.01, condition1 := P_On, Neglect1 := 0.07, ALARMDELAY := #200, RESETDELAY := #400, out1 => W201.06)  ; 灌装原位报警条件, 灌装缸原位, 灌装缸原位异常

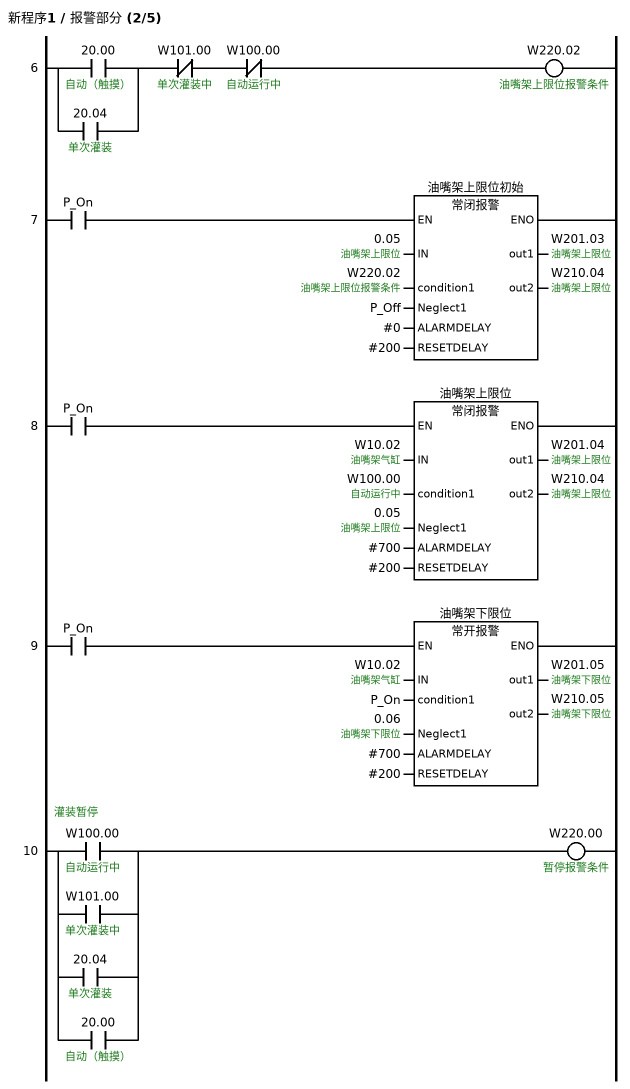
; rung 6
LD 20.00  ; 自动（触摸）
OR 20.04  ; 单次灌装
ANDNOT W101.00  ; 单次灌装中
ANDNOT W100.00  ; 自动运行中
OUT W220.02  ; 油嘴架上限位报警条件
; rung 7
LD P_On
CALL 油嘴架上限位初始 : 常闭报警 (IN := 0.05, condition1 := W220.02, Neglect1 := P_Off, ALARMDELAY := #0, RESETDELAY := #200, out1 => W201.03, out2 => W210.04)  ; 油嘴架上限位, 油嘴架上限位报警条件
; rung 8
LD P_On
CALL 油嘴架上限位 : 常闭报警 (IN := W10.02, condition1 := W100.00, Neglect1 := 0.05, ALARMDELAY := #700, RESETDELAY := #200, out1 => W201.04, out2 => W210.04)  ; 油嘴架气缸, 自动运行中, 油嘴架上限位
; rung 9
LD P_On
CALL 油嘴架下限位 : 常开报警 (IN := W10.02, condition1 := P_On, Neglect1 := 0.06, ALARMDELAY := #700, RESETDELAY := #200, out1 => W201.05, out2 => W210.05)  ; 油嘴架气缸, 油嘴架下限位
; rung 10: 灌装暂停
LD W100.00  ; 自动运行中
OR W101.00  ; 单次灌装中
OR 20.04  ; 单次灌装
OR 20.00  ; 自动（触摸）
OUT W220.00  ; 暂停报警条件

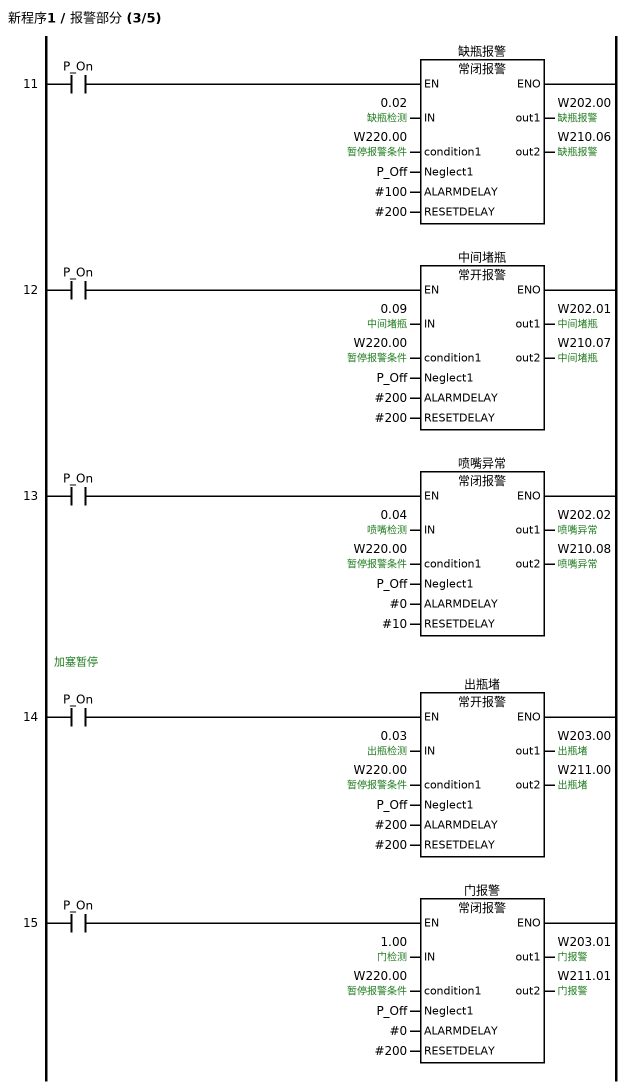
; rung 11
LD P_On
CALL 缺瓶报警 : 常闭报警 (IN := 0.02, condition1 := W220.00, Neglect1 := P_Off, ALARMDELAY := #100, RESETDELAY := #200, out1 => W202.00, out2 => W210.06)  ; 缺瓶检测, 暂停报警条件, 缺瓶报警
; rung 12
LD P_On
CALL 中间堵瓶 : 常开报警 (IN := 0.09, condition1 := W220.00, Neglect1 := P_Off, ALARMDELAY := #200, RESETDELAY := #200, out1 => W202.01, out2 => W210.07)  ; 中间堵瓶, 暂停报警条件
; rung 13
LD P_On
CALL 喷嘴异常 : 常闭报警 (IN := 0.04, condition1 := W220.00, Neglect1 := P_Off, ALARMDELAY := #0, RESETDELAY := #10, out1 => W202.02, out2 => W210.08)  ; 喷嘴检测, 暂停报警条件, 喷嘴异常
; rung 14: 加塞暂停
LD P_On
CALL 出瓶堵 : 常开报警 (IN := 0.03, condition1 := W220.00, Neglect1 := P_Off, ALARMDELAY := #200, RESETDELAY := #200, out1 => W203.00, out2 => W211.00)  ; 出瓶检测, 暂停报警条件, 出瓶堵
; rung 15
LD P_On
CALL 门报警 : 常闭报警 (IN := 1.00, condition1 := W220.00, Neglect1 := P_Off, ALARMDELAY := #0, RESETDELAY := #200, out1 => W203.01, out2 => W211.01)  ; 门检测, 暂停报警条件, 门报警

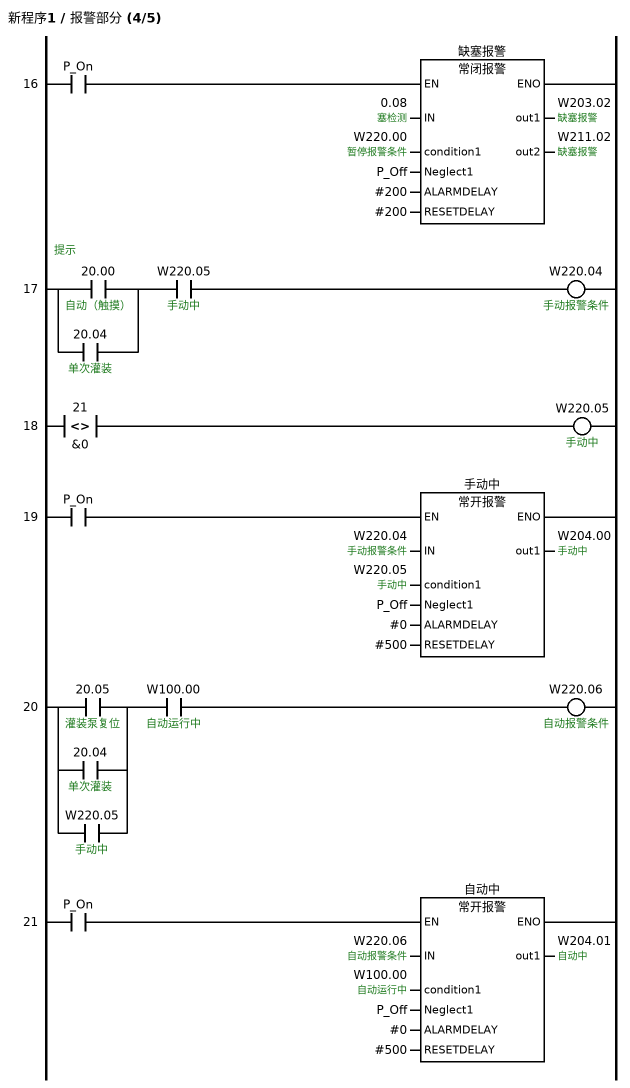
; rung 16
LD P_On
CALL 缺塞报警 : 常闭报警 (IN := 0.08, condition1 := W220.00, Neglect1 := P_Off, ALARMDELAY := #200, RESETDELAY := #200, out1 => W203.02, out2 => W211.02)  ; 塞检测, 暂停报警条件, 缺塞报警
; rung 17: 提示
LD 20.00  ; 自动（触摸）
OR 20.04  ; 单次灌装
AND W220.05  ; 手动中
OUT W220.04  ; 手动报警条件
; rung 18
LD<>L(306) 21 &0
OUT W220.05  ; 手动中
; rung 19
LD P_On
CALL 手动中 : 常开报警 (IN := W220.04, condition1 := W220.05, Neglect1 := P_Off, ALARMDELAY := #0, RESETDELAY := #500, out1 => W204.00)  ; 手动报警条件, 手动中
; rung 20
LD 20.05  ; 灌装泵复位
OR 20.04  ; 单次灌装
OR W220.05  ; 手动中
AND W100.00  ; 自动运行中
OUT W220.06  ; 自动报警条件
; rung 21
LD P_On
CALL 自动中 : 常开报警 (IN := W220.06, condition1 := W100.00, Neglect1 := P_Off, ALARMDELAY := #0, RESETDELAY := #500, out1 => W204.01)  ; 自动报警条件, 自动运行中, 自动中

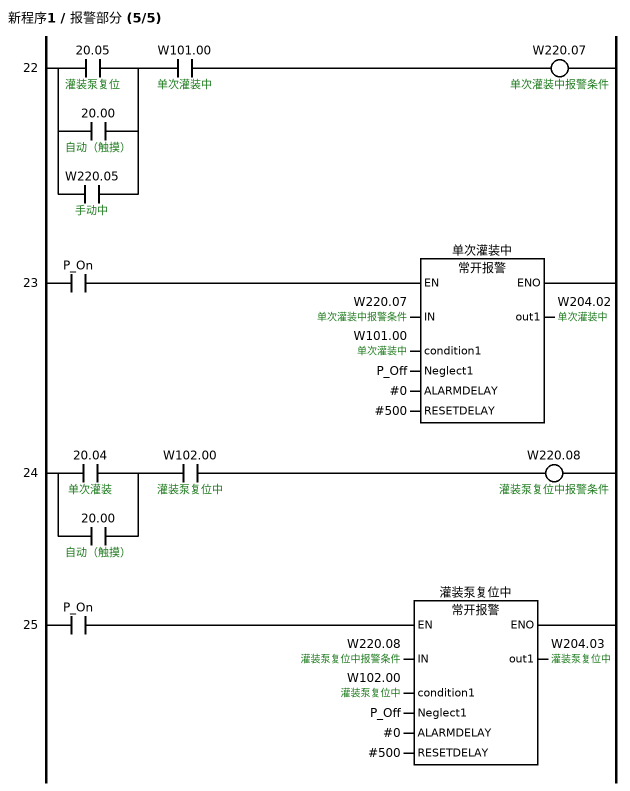
; rung 22
LD 20.05  ; 灌装泵复位
OR 20.00  ; 自动（触摸）
OR W220.05  ; 手动中
AND W101.00  ; 单次灌装中
OUT W220.07  ; 单次灌装中报警条件
; rung 23
LD P_On
CALL 单次灌装中 : 常开报警 (IN := W220.07, condition1 := W101.00, Neglect1 := P_Off, ALARMDELAY := #0, RESETDELAY := #500, out1 => W204.02)  ; 单次灌装中报警条件, 单次灌装中
; rung 24
LD 20.04  ; 单次灌装
OR 20.00  ; 自动（触摸）
AND W102.00  ; 灌装泵复位中
OUT W220.08  ; 灌装泵复位中报警条件
; rung 25
LD P_On
CALL 灌装泵复位中 : 常开报警 (IN := W220.08, condition1 := W102.00, Neglect1 := P_Off, ALARMDELAY := #0, RESETDELAY := #500, out1 => W204.03)  ; 灌装泵复位中报警条件, 灌装泵复位中

### Section 保存调用

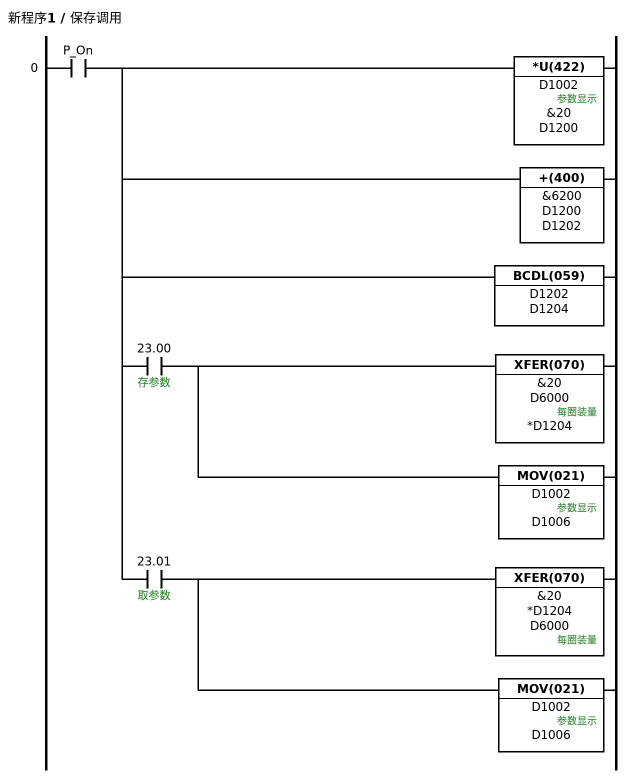
; rung 0
LD P_On
OUT TR0
*U(422) D1002 &20 D1200  ; 参数显示
+(400) &6200 D1200 D1202
BCDL(059) D1202 D1204
AND 23.00  ; 存参数
XFER(070) &20 D6000 *D1204  ; 每圈装量
MOV(021) D1002 D1006  ; 参数显示
LD TR0
AND 23.01  ; 取参数
XFER(070) &20 *D1204 D6000  ; 每圈装量
MOV(021) D1002 D1006  ; 参数显示

### Section END
; rung 0
END(001)

## Function block 常闭报警
VAR_INPUT
  IN : BOOL;
  condition1 : BOOL;  (* 报警条件1 *)
  Neglect1 : BOOL;
  ALARMDELAY : WORD;  (* 报警延时 *)
  RESETDELAY : WORD;  (* 恢复延时 *)
END_VAR
VAR_OUTPUT
  out1 : BOOL;  (* 报警输出 *)
  out2 : BOOL;
END_VAR
VAR
  TM1 : TIMER;
  TM2 : TIMER;
END_VAR

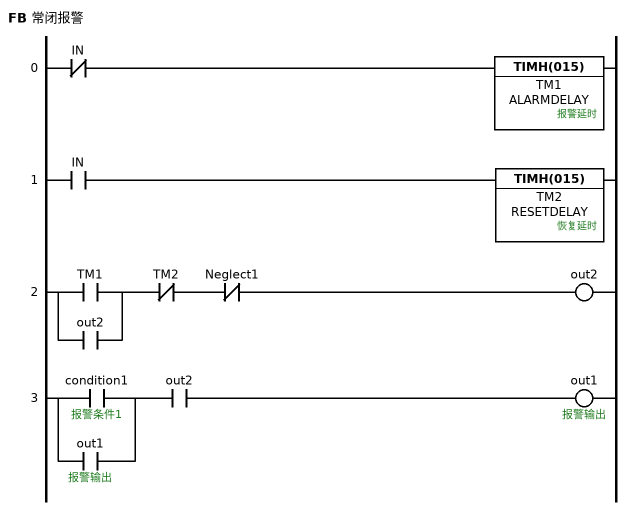
; rung 0
LDNOT IN
TIMH(015) TM1 ALARMDELAY  ; 报警延时
; rung 1
LD IN
TIMH(015) TM2 RESETDELAY  ; 恢复延时
; rung 2
LD TM1
OR out2
ANDNOT TM2
ANDNOT Neglect1
OUT out2
; rung 3
LD condition1  ; 报警条件1
OR out1  ; 报警输出
AND out2
OUT out1  ; 报警输出

## Function block 常开报警
VAR_INPUT
  IN : BOOL;
  condition1 : BOOL;  (* 报警条件1 *)
  Neglect1 : BOOL;
  ALARMDELAY : WORD;  (* 报警延时 *)
  RESETDELAY : WORD;  (* 恢复延时 *)
END_VAR
VAR_OUTPUT
  out1 : BOOL;  (* 报警输出 *)
  out2 : BOOL;
END_VAR
VAR
  TM1 : TIMER;
  TM2 : TIMER;
END_VAR

